FUNCTION_BLOCK ADI_TO_ALI (* Composite FB for converting ADI (DINT) adapter to ALI (LINT) adapter — numeric conversion (value-preserving cast; narrowing may truncate, widening/sign-extension is safe). *)
  (* Standard: 61499-2; Description: Copyright (c) 2026 HR Agrartechnik GmbH This program and the accompanying materials are made available under the terms of the Eclipse Public License 2.0 which is available at https://www.eclipse.org/legal/epl-2.0/ SPDX-License-Identifier: EPL-2.0 *)
  (* Version 1.0, 2026-02-17, Franz Höpfinger, HR Agrartechnik GmbH *)
  PACKAGE adapter::conversion::unidirectional;
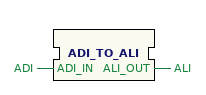
  SOCKETS
    ADI_IN : adapter::types::unidirectional::ADI; (* DINT Adapter Input *)
  END_SOCKETS
  PLUGS
    ALI_OUT : adapter::types::unidirectional::ALI; (* LINT Adapter Output *)
  END_PLUGS
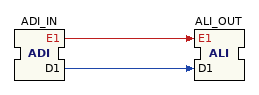
  EVENT_CONNECTIONS
    ADI_IN.E1 TO ALI_OUT.E1;
  END_CONNECTIONS
  DATA_CONNECTIONS
    ADI_IN.D1 TO ALI_OUT.D1;
  END_CONNECTIONS
END_FUNCTION_BLOCK
